# EPICS autosave request: axisSXR40App/Db/axisSXR40_settings.req
$(P)$(R)BitDepth
$(P)$(R)FrameSpeed
$(P)$(R)BitDepth
$(P)$(R)BinMode
$(P)$(R)GainMode
$(P)$(R)AutoExposure
$(P)$(R)FanGear
$(P)$(R)AutoLevels
$(P)$(R)Histogram
$(P)$(R)Enhance
$(P)$(R)DefectCorrection
$(P)$(R)EnableDenoise
$(P)$(R)FlatCorrection
$(P)$(R)DynRgeCorrection
$(P)$(R)FrameFormat
$(P)$(R)Brightness
$(P)$(R)BlackLevel
$(P)$(R)Sharpness
$(P)$(R)NoiseLevel
$(P)$(R)HDRK
$(P)$(R)Gamma
$(P)$(R)Contrast
$(P)$(R)LeftLevels
$(P)$(R)RightLevels
$(P)$(R)TriggerEdge
$(P)$(R)TriggerExposure
$(P)$(R)TriggerDelay
$(P)$(R)TriggerOut1Mode
$(P)$(R)TriggerOut1Edge
$(P)$(R)TriggerOut1Delay
$(P)$(R)TriggerOut1Width
$(P)$(R)TriggerOut2Mode
$(P)$(R)TriggerOut2Edge
$(P)$(R)TriggerOut2Delay
$(P)$(R)TriggerOut2Width
$(P)$(R)TriggerOut3Mode
$(P)$(R)TriggerOut3Edge
$(P)$(R)TriggerOut3Delay
$(P)$(R)TriggerOut3Width

# TECEnable is deliberately NOT saved here, and must not be added.
#
# The record is PINI=YES with a default of Disable, so every boot writes the TEC
# OFF -- the safe state, and the only state software can justify, since nothing
# here can see the coolant loop (see the HAZARD note in axisSXR40.template).
# Autosaving it would invert that: a session that left the TEC enabled would
# silently re-enable it at the next boot, unattended, with no confirmation that
# water is flowing. The manual states a water failure can damage the sensor.
# Leave it out.

file "ADBase_settings.req", P=$(P), R=$(R)
